# EPICS autosave request: roles/install_ioc/tasks/device_types/tetramm/files/auto_settings.req
file "quadEM_settings.req", P=$(P), R=
file "quadEM_Plugin_settings.req", P=$(P), R=
# file "quadEM_TimeSeries_settings.req", P=$(P), R=
